PROGRAM MAIN
VAR

inc1 : DINT := 0;

END_VAR

GVL.mOutTrain := GVL.mInTrain;

FOR inc1 := 0 TO 150 DO
	//Sets Red Lights
	IF GVL.mInOccupancies[inc1] = 0
	THEN
		GVL.mOutLeftLights[inc1] := 0;
		GVL.mOutRightLights[inc1] := 0;
	//Sets green lights
	ELSE
		GVL.mOutLeftLights[inc1] := 2;
		GVL.mOutRightLights[inc1] := 2;
	END_IF
END_FOR

FOR inc1 := 1 TO 149 DO
	//Sets Yellow Lights
	IF GVL.mInOccupancies[inc1-1] = 0 AND GVL.mInOccupancies[inc1] <> 0
	THEN
		GVL.mOutRightLights[inc1] := 1;
	END_IF
	IF GVL.mInOccupancies[inc1+1] = 0 AND GVL.mInOccupancies[inc1] <> 0
	THEN
	GVL.mOutLeftLights[inc1] := 1;
	END_IF
END_FOR

//0 to 61 corresponds to blocks 1 to 62
//76 to 150 corresponds to 

FOR inc1 := 0 TO 150 DO
	
	GVL.mOutOccupancies[inc1] := GVL.mInOccupancies[inc1];
	GVL.mOutSpeeds[inc1] := GVL.mInSpeeds[inc1];
	GVL.mOutAuthorities[inc1] := GVL.mInAuthorities[inc1];
	GVL.mOutMaintenance[inc1] := GVL.mInMaintenance[inc1];
	IF GVL.mInSpeeds[inc1] < GVL.mSpeedLimits[inc1]
	THEN
		GVL.mOutSpeeds[inc1] := GVL.mInSpeeds[inc1];
	ELSE
		GVL.mOutSpeeds[inc1] := GVL.mSpeedLimits[inc1];
	END_IF

END_FOR

inc1 := 0;

//This starts the main track logic section

//Crossing Logic
IF GVL.mInOccupancies[18] = 0 THEN
	GVL.mOutCrossings[18] := 1;
ELSE
	GVL.mOutCrossings[18] := 0;
END_IF


//Switch Logic

//Set switch on block 13
IF GVL.mInMaintenance[12] = 1 THEN
    GVL.mOutSwitch[12] := GVL.mInSwitch[12];
ELSE
    IF GVL.mInOccupancies[11] = 0 THEN
    	GVL.mOutSwitch[12] := 11;
    ELSE
		GVL.mOutSwitch[12] := 0;
	END_IF
END_IF

//Set switch on block 29
IF GVL.mInMaintenance[28] = 1 THEN
    GVL.mOutSwitch[28] := GVL.mInSwitch[28];
ELSE
    IF GVL.mInOccupancies[28] = 0 THEN
    FOR inc1 := 12 TO 28 DO 
        IF GVL.mInOccupancies[inc1] = 0 THEN
            GVL.mOutSwitch[28] := 149;
            Exit;
        ELSE 
            GVL.mOutSwitch[28] := 29;
        END_IF
    END_FOR
	END_IF
END_IF


//Set switch on block 58
IF GVL.mInMaintenance[57] = 1 THEN
    GVL.mOutSwitch[57] := GVL.mInSwitch[57];
ELSE
	GVL.mOutSwitch[57] := 58;
END_IF
	
//Set switch on block
IF GVL.mInMaintenance[76] = 1 THEN
    GVL.mOutSwitch[76] := GVL.mInSwitch[76];
ELSE
    IF GVL.mInOccupancies[75] = 0 THEN
    FOR inc1 := 76 TO 84 DO 
        IF GVL.mInOccupancies[inc1] = 0 THEN
            GVL.mOutSwitch[75] := 100;
            Exit;
        ELSE 
            GVL.mOutSwitch[75] := 74;
        END_IF
    END_FOR
	END_IF
END_IF

IF GVL.mInMaintenance[84] = 1 THEN
    GVL.mOutSwitch[84] := GVL.mInSwitch[84];
ELSE
    IF GVL.mInOccupancies[99] = 0 THEN
    FOR inc1 := 76 TO 84 DO 
        IF GVL.mInOccupancies[inc1] = 0 THEN
            GVL.mOutSwitch[84] := 85;
            Exit;
        ELSE 
            GVL.mOutSwitch[84] := 99;
        END_IF
    END_FOR
	END_IF
END_IF

END_PROGRAM

(* stored: Version 1.1.0.1, ProductVersion 3.1.4024.11
   POU MAIN: Id {4c8b3e77-e4d8-438f-9dd4-fa42d08617c7}, SpecialFunc None *)
